{attribute 'linkalways'} 
{attribute 'no_explicit_call' := 'This FB is a CLASS and must be accessed using methods or properties'}
{attribute 'enable_dynamic_creation'}
FUNCTION_BLOCK FINAL SEL_BYTE EXTENDS Node
VAR
	g : _BOOL(FALSE);
	in1 : _BYTE(0);
	in2 : _BYTE(0);
	out : _BYTE(0);
END_VAR

METHOD PUBLIC Clone : I_Node
VAR
	pNode : POINTER TO SEL_BYTE;
END_VAR
pNode := __NEW(SEL_BYTE);
Clone := pNode^;
END_METHOD

METHOD FB_init : BOOL
VAR_INPUT
	bInitRetains : BOOL; // if TRUE, the retain variables are initialized (warm start / cold start)
	bInCopyCode : BOOL;  // if TRUE, the instance afterwards gets moved into the copy code (online change)
END_VAR
AddInput('g',THIS^.g);
AddInput('in1',THIS^.in1);
AddInput('in2',THIS^.in2);
AddOutput('out', THIS^.out);
END_METHOD

METHOD PROTECTED OnExecute
VAR
END_VAR
IF g.value THEN
	out.value := in2.value;
ELSE
	out.value := in1.value;
END_IF
END_METHOD

END_FUNCTION_BLOCK

(* stored: Version 1.1.0.1, ProductVersion 3.1.4024.15
   POU SEL_BYTE: Id {e60af96b-011e-4829-b885-99fffc55a9a9}, SpecialFunc None
   Folder Constructor: Id {77cfc530-66b1-4c49-88d7-20517b8b304a}
   Method Clone: Id {fc17124e-cacb-4197-9230-2fc2a085f060}
   Method FB_init: Id {6293d7d0-a075-4e84-854f-b7ac17e9cf59}
   Method OnExecute: Id {2094e714-a903-4ef7-b9ec-420afbb2fe0a} *)
